FUNCTION_BLOCK CommonBase
VAR_INPUT
END_VAR
VAR_OUTPUT
END_VAR
VAR
	default : int := 16#ff; //for base class , minimun requires one field to locate address
END_VAR

METHOD ConfigureRead : CellDataBlock
VAR_INPUT
END_VAR
END_METHOD

METHOD ConfigureWrite : BOOL
VAR_INPUT
	input : CellDataBlock;
END_VAR
END_METHOD

METHOD Control : BOOL
VAR_INPUT
	input : CellDataBlock;
	mode : eModes;
END_VAR
END_METHOD

METHOD ErrorClear : BOOL
VAR_INPUT
	input : eErrorClearWays;
END_VAR
END_METHOD

METHOD ErrorDetect : int
VAR_INPUT
END_VAR
END_METHOD

METHOD Monitor : CellDataBlock
VAR_INPUT
END_VAR
END_METHOD

METHOD Stop : BOOL
VAR_INPUT
END_VAR
END_METHOD

METHOD TypeCode : eCategrories
VAR_INPUT
END_VAR
END_METHOD

END_FUNCTION_BLOCK

(* stored: Version 1.1.0.1, ProductVersion 3.1.4022.10
   POU CommonBase: Id {0ec98e57-59b2-46ad-8038-cac0ed0e74a9}, SpecialFunc None
   Method ConfigureRead: Id {8e0df28b-cbcb-4f0b-9e41-e6a240ff5ddf}
   Method ConfigureWrite: Id {ae3bac82-ca4b-49e7-bb0c-2ffd48d7a2d3}
   Method Control: Id {6b2845e0-d489-487e-a42c-42934f1729db}
   Method ErrorClear: Id {b26b719e-f527-4ef0-bd52-663bd6511afd}
   Method ErrorDetect: Id {f95a086f-f03e-4047-a51e-55e0cdb1901d}
   Method Monitor: Id {6e2674a7-55cf-4f68-b8fc-bd23a5a9c826}
   Method Stop: Id {23e1061a-1dcf-48fd-bd32-abbb323b4a0b}
   Method TypeCode: Id {e730d55b-d0ba-4b79-ae5c-fc301e130191} *)
